// TIA Portal V16 export
// export: Created 2022-03-28T07:44:09.282286Z, ExportSetting WithDefaults, DisplayName Totally Integrated Automation Portal, DisplayVersion V16 Update 5, DisplayName TIA Portal Version Control Interface, DisplayVersion V16 Update 2, DisplayName TIA Portal Openness, DisplayVersion V16 Update 5, DisplayName STEP 7 Professional, DisplayVersion V16 Update 5, DisplayName STEP 7 Safety, DisplayVersion V16, DisplayName WinCC Professional, DisplayVersion V16 Update 5
TYPE "udtCounters"
// stored: IsFailsafeCompliant false
   STRUCT
      diPreselectionValue : DInt;
      diTotalOK : DInt;
      diPartialOK : DInt;
      diConsecutiveOK : DInt;
      diTotalNOK : DInt;
      diPartialNOK : DInt;
      diConsecutiveNOK : DInt;
      diScrapBox : DInt;
      stSettings : Struct
         diScrapBoxSize : DInt;
         diNOKValueToBlock : DInt;
         diOKValueToResetNOK : DInt;
      END_STRUCT;
      stButtons : Struct
         bResetTotalOK : Bool;
         bResetPartialOK : Bool;
         bResetConsecutiveOK : Bool;
         bResetTotalNOK : Bool;
         bResetPartialNOK : Bool;
         bResetConsecutiveNOK : Bool;
         bResetScrapBox : Bool;
      END_STRUCT;
   END_STRUCT;
END_TYPE
